(* CODESYS project CODESYS_TEST

Project tree, tasks and I/O mapping:
  _750_8210_PFC200 : 750-8210 PFC200, WAGO, order no. 750-8210, version 6.3.0.12
    application Application
    Kbus : Kbus, WAGO, version 2.1.0.1
        unmapped channels: K-BUS diagnostics
  Device : CODESYS Control Win V3, 3S - Smart Software Solutions GmbH, version 3.5.19.70
    application Application
      libraries: Standard, 3.5.18.0 (System)
      task MainTask (cyclic, interval t#20ms, priority 1) calls PLC_PRG
      program PLC_PRG [ST]
      program POU_1 [UML]: POU_1_State1_DO
      program POU [FBD]
      program test [FBD]
*)

// Device/Application/PLC_PRG
PROGRAM PLC_PRG
VAR
END_VAR

END_PROGRAM

// Device/Application/POU_1
PROGRAM POU_1
VAR
END_VAR

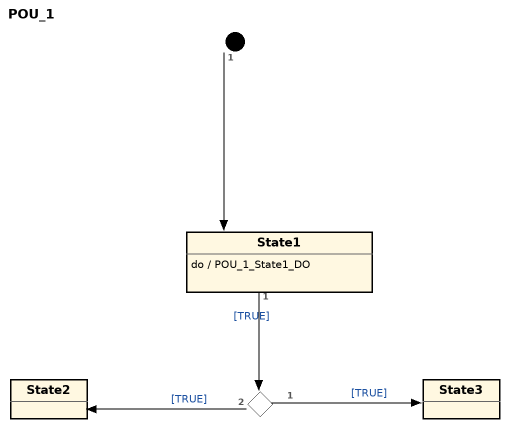
STATECHART POU_1  // abortable
    START StartState1
    STATE State1
        do / POU_1_State1_DO
    STATE State2
    CHOICE ChoiceElement1
    STATE State3
    StartState1 -> State1  // priority 1, on completion
    State1 -> ChoiceElement1 [TRUE] // priority 1
    ChoiceElement1 -> State3 [TRUE] // priority 1
    ChoiceElement1 -> State2 [TRUE] // priority 2
END_STATECHART

ACTION POU_1_State1_DO:

END_ACTION

END_PROGRAM

// Device/Application/POU
PROGRAM POU
VAR
END_VAR

// NETWORK 1

END_PROGRAM

// Device/Application/test
PROGRAM test
VAR
END_VAR

// NETWORK 1

END_PROGRAM
